FUNCTION_BLOCK XtsClassTestSuite
VAR
	
END_VAR

END_FUNCTION_BLOCK

(* stored: Version 1.1.0.1
   POU XtsClassTestSuite: Id {7d78b050-bb38-4110-9cb6-9104c4069eaf}, SpecialFunc None *)
